		// If no next zone or function is available
		IF NextTransportData.eFunctionNumber = E_FunctionNumber.F_BEGIN_FUNCTION AND
		   Param.reNextFunctionNumber = E_FunctionNumber.F_BEGIN_FUNCTION THEN	
			// Update for this transport valid trasport parameter
			TransportParam := ZoneData.TransportControlData.TransportParam;	
		END_IF

		// If zone is occupied
		IF ZoneOccupiedSignal THEN
			// Reset clearing
			fbClearing(Run := FALSE);
			// Reset delay zone free
			fbDelayZoneFree(Run := FALSE);

			// If not status occupied
			IF NOT ZoneData.TransportControlData.Occupied THEN
				DelayDistance := TransportParam.StopDelayDistance - StoppingDistance;
				
				IF DelayDistance < 0 THEN
					DelayDistance := 0;
				END_IF
				
				// Run delay zone occupied
				fbDelayZoneOccupied(
					Run					:= TRUE,
					EncoderValueInc		:= EncoderValue,
					MaxEncoderValueInc	:= MaxEncoderValue,
					RateIncPerMM		:= 1,
					SetPoint			:= DelayDistance);

				// Set status occupied	
				IF fbDelayZoneOccupied.Q THEN
					DriveMultiTU_Run := FALSE;
					fbDelayZoneOccupied(RUN := FALSE);
					fbClearing(Run := FALSE);
					ZoneData.TransportControlData.Occupied := TRUE;
					ZoneData.TransportControlData.eTransportState := E_TransportState.MULTI_TU_OCCUPIED;
				END_IF					

			// Switch to occupied state if handover is not active
			ELSIF ZoneData.TransportControlData.eHandOverState <> E_HandOverState.ACTIVE THEN
				DriveMultiTU_Run := FALSE;
				ZoneData.TransportControlData.eTransportState := E_TransportState.MULTI_TU_OCCUPIED;
			END_IF
		
		// Zone is not occupied	
		ELSE
			// Reset delay zone occupied
			fbDelayZoneOccupied(RUN := FALSE);		

			// If status occupied
			IF ZoneData.TransportControlData.Occupied THEN
				// If handover is active
				IF ZoneData.TransportControlData.eHandOverState = E_HandOverState.ACTIVE THEN
					DelayDistance := TransportParam.ZoneEndLength - StoppingDistance;
					
					IF DelayDistance < 0 THEN
						DelayDistance := 0;
					END_IF
					
					// Run delay zone free
					fbDelayZoneFree(
						Run					:= TRUE,
						EncoderValueInc		:= EncoderValue,
						MaxEncoderValueInc	:= MaxEncoderValue,
						RateIncPerMM		:= 1,
						SetPoint			:= DelayDistance);
	
					// Restet status occupied if zone is free during handover
					IF fbDelayZoneFree.Q THEN
						fbDelayZoneFree(Run := FALSE);
						ZoneData.TransportControlData.Occupied := FALSE;
					END_IF
				ELSE
					// Switch to occupied state if handover is not active
					DriveMultiTU_Run := FALSE;
					fbDelayZoneFree(Run := FALSE);
					ZoneData.TransportControlData.eTransportState := E_TransportState.MULTI_TU_OCCUPIED;
				END_IF
	
			// Status is not occupied
			ELSE
				// Reset clearing if takeover is active
				IF ZoneData.TransportControlData.eTakeOverState = E_TakeOverState.ACTIVE THEN
					fbClearing(Run := FALSE);	
				ELSE
					// Run clearing
					fbClearing(
						Run					:= TRUE,
						EncoderValueInc		:= EncoderValue,
						MaxEncoderValueInc	:= MaxEncoderValue,
						RateIncPerMM		:= 1,
						SetPoint			:= Param.rSettings.ClearingDistance);
	
					// Switch to state free if zone is clear
					IF fbClearing.Q THEN
						DriveMultiTU_Run := FALSE;
						fbClearing(Run := FALSE);
						ZoneData.TransportControlData.NumberOfPresentTUs := 0;
						ZoneData.TransportControlData.eTransportState := E_TransportState.FREE;
					END_IF
				END_IF
			END_IF
		END_IF

(*************************************************************************
  Multi TU Occupied
*************************************************************************)
	E_TransportState.MULTI_TU_OCCUPIED:		
		// Request next zone for handover
		M_RequestNext();

		// If next zone is available
		IF NextTransportData.eFunctionNumber <> E_FunctionNumber.F_BEGIN_FUNCTION THEN
			// If handover is active
			IF ZoneData.TransportControlData.eHandOverState = E_HandOverState.ACTIVE THEN
				ZoneData.TransportControlData.eTransportState := E_TransportState.MULTI_TU;
			END_IF
		ELSE
			// Update for this transport valid trasport parameter
			TransportParam := ZoneData.TransportControlData.TransportParam;
		END_IF

		// If the occupied state needs not to be latched
		IF NOT Param.rSettings.EnableLatchOccupiedState THEN		
			// If zone is free
			IF NOT ZoneOccupiedSignal THEN
				// Run occupied free timer
				fbZoneOccupiedFreeTimer(IN := TRUE, PT := tZoneFree);

				// Zone is free without transfer
				IF fbZoneOccupiedFreeTimer.Q THEN
					fbZoneOccupiedFreeTimer(IN := FALSE);
					ZoneData.TransportControlData.Occupied := FALSE;
					TransportTrspDataReq.DeleteNextTransportData := TRUE;
	
					// Update number of present TUs
					IF ZoneData.TransportControlData.NumberOfPresentTUs > 0 THEN
						ZoneData.TransportControlData.NumberOfPresentTUs := ZoneData.TransportControlData.NumberOfPresentTUs -1;	
					END_IF			
	
					ZoneData.TransportControlData.eTransportState := E_TransportState.MULTI_TU;
				END_IF	
			ELSE
				// Reset occupied free timer
				fbZoneOccupiedFreeTimer(IN := FALSE);
			END_IF
		END_IF
				
(*************************************************************************
  Multi TU Stop
*************************************************************************)
	E_TransportState.MULTI_TU_STOP:
		// If function is started
		IF Param.rOperationState.eState = E_PositionState.STARTED THEN
			// If transport is enabled
			IF Inputs.Enable.Transport THEN		
				// If no error is active
				IF ErrorData.ErrorType <> E_ErrorType.ERROR THEN
					// If take and handover is not interrupted
					IF  ZoneData.TransportControlData.eTakeOverState <> E_TakeOverState.INTERRUPTED AND
                        ZoneData.TransportControlData.eHandOverState <> E_HandOverState.INTERRUPTED THEN
						fbZoneOccupiedFreeTimer(IN := FALSE);
						// Resume to multi TU
						ZoneData.TransportControlData.eTransportState := E_TransportState.MULTI_TU;
					END_IF
				END_IF
			END_IF
		END_IF
		
(*************************************************************************
  Simultaneous
*************************************************************************)
	E_TransportState.SIMULTANEOUS:
		// Swich to simultaneous stop if take or handover is stop or interrupted
		IF ZoneData.TransportControlData.eTakeOverState = E_TakeOverState.STOP OR 
           ZoneData.TransportControlData.eHandOverState = E_HandOverState.STOP OR
		   ZoneData.TransportControlData.eTakeOverState = E_TakeOverState.INTERRUPTED OR
		   ZoneData.TransportControlData.eHandOverState = E_HandOverState.INTERRUPTED THEN
		    DriveFeedInRun := FALSE;
			ZoneData.TransportControlData.eTransportState := E_TransportState.SIMULTANEOUS_STOP;
		END_IF	

		// If zone is physically occupied
		IF ZoneOccupiedSignal THEN
			// Reset timeout take
			fbTimeoutTake(Run := FALSE);
			// Reset delay zone free
			fbDelayZoneFree(Run := FALSE);

			// If zone is logically not occupied,
			// -> move forward until logically occupied 
			IF NOT ZoneData.TransportControlData.Occupied THEN
				// Set drive on
				DriveFeedInRun := TRUE;

				DelayDistance := TransportParam.StopDelayDistance - StoppingDistance;
				
				IF DelayDistance < 0 THEN
					DelayDistance := 0;
				END_IF
				
				// Run delay zone occupied
				fbDelayZoneOccupied(
					Run					:= TRUE,
					EncoderValueInc		:= EncoderValue,
					MaxEncoderValueInc	:= MaxEncoderValue,
					RateIncPerMM		:= 1,
					SetPoint			:= DelayDistance);

				// Set status occupied	
				IF fbDelayZoneOccupied.Q THEN
					fbDelayZoneOccupied(RUN := FALSE);
					fbClearing(Run := FALSE);
					ZoneData.TransportControlData.Occupied := TRUE;
				END_IF					
		
			// Switch to simultaneous occupied state if handover is not active
			ELSIF ZoneData.TransportControlData.eHandOverState <> E_HandOverState.ACTIVE THEN 
				DriveFeedInRun := FALSE;
				ZoneData.TransportControlData.eTransportState := E_TransportState.SIMULTANEOUS_OCCUPIED;
			ELSE
				DriveFeedInRun := FALSE;
			END_IF			
			
		// Zone is physically not occupied	
		ELSE
			// Reset delay zone occupied
			fbDelayZoneOccupied(RUN := FALSE);		

			// If zone is logically occupied
			IF ZoneData.TransportControlData.Occupied THEN
				// If handover is active
				IF ZoneData.TransportControlData.eHandOverState = E_HandOverState.ACTIVE THEN
					DelayDistance := TransportParam.ZoneEndLength - StoppingDistance;
                    DriveFeedInRun := TRUE;
					
					IF DelayDistance < 0 THEN
						DelayDistance := 0;
					END_IF
					
					// Run delay zone free
					fbDelayZoneFree(
						Run					:= TRUE,
						EncoderValueInc		:= EncoderValue,
						MaxEncoderValueInc	:= MaxEncoderValue,
						RateIncPerMM		:= 1,
						SetPoint			:= DelayDistance);
	
					// Restet status occupied if zone is free during handover
					IF fbDelayZoneFree.Q THEN
						fbDelayZoneFree(Run := FALSE);
						ZoneData.TransportControlData.Occupied := FALSE;
					END_IF
				ELSE
					// Switch to occupied state if handover is not active
					DriveFeedInRun := FALSE;
					fbDelayZoneFree(Run := FALSE);
					ZoneData.TransportControlData.eTransportState := E_TransportState.SIMULTANEOUS_OCCUPIED;
				END_IF
	
			// Zone is logically not occupied -> (Feedin)
			// adption to BCF 1.13 where this only occure if MFC is disabled
			ELSIF(NOT Param.rSettings.EnableMFC) THEN
				// Set drive on
				DriveFeedInRun := TRUE;
				
				// Timeout take monitoring
				IF Param.rSettings.TimeoutTakeDistance <> 0 THEN
					TimeoutTakeDistance := Param.rSettings.TimeoutTakeDistance;
				ELSE
					TimeoutTakeDistance := (UINT_TO_DINT(TransportParam.ZoneLength)
											- TransportParam.ZoneEndLength
											+ TransportParam.StopDelayDistance
											+ PrevTransportParam.ZoneEndLength) * TIMEOUT_TAKE_FACTOR;
				END_IF			
				
				IF TimeoutTakeDistance < 0 THEN
					TimeoutTakeDistance := 0;
				END_IF
				
				// Run timeout take
				fbTimeoutTake(
					Run					:= TRUE,
					EncoderValueInc		:= EncoderValue,
					MaxEncoderValueInc	:= MaxEncoderValue,
					SetPoint			:= TimeoutTakeDistance);
							
				// If timeout take, clear TU-data index and end feed in
				IF fbTimeoutTake.Q THEN
					// Debug message: '11-001-0095-01-1,  TU_DataIndex of implausible simultaneously takeover deleted,  TU_DataIndex = 12345,  TuID = 112233,  AssignmentID = 12345678'
					DebugMsg := '';
					DebugMsg := CONCAT(DebugMsg, F_AddDividerToSisString(Param.rSettings.ZoneName));
					DebugMsg := CONCAT(DebugMsg, ',  TU_DataIndex of implausible simultaneously takeover deleted');
					DebugMsg := CONCAT(DebugMsg, F_CreateTU_DataString(ZoneData.TransportControlData.TU_DataIndex));
					fbDebugMsg.M_SendErrorMsg(DebugMsg);
					
					DriveFeedInRun := FALSE;
					fbTimeoutTake(Run := FALSE);
					fbDelayZoneOccupied(Run := FALSE);
					M_DeleteTU_DataIndex(mSendTUR := TRUE);
					TransportTrspDataReq.DeleteNextTransportData := TRUE;
					ZoneData.TransportControlData.NumberOfPresentTUs := 0;	
	
					// If free run is enable
					IF Param.rSettings.EnableFreeRun THEN
						DriveFreeRun := TRUE;
						ZoneData.TransportControlData.eTransportState := E_TransportState.FREE_RUN;
					ELSE
						ZoneData.TransportControlData.eTransportState := E_TransportState.FREE;	
					END_IF
				END_IF
			END_IF
		END_IF
		
(*************************************************************************
  Simultaneous Occupied
*************************************************************************)
	E_TransportState.SIMULTANEOUS_OCCUPIED:		
		// If simultaneous transport is disable, switch to basic transport
		IF NOT Param.rSettings.EnableSimultaneousTransport AND
			NOT ZoneData.AddOn.Orders.EnableSimultaneousTransport THEN
			ZoneData.TransportControlData.eTransportState := E_TransportState.OCCUPIED;
		END_IF
			
		// Request prev zone for takeover
		M_RequestPrev();

		// Request next zone for handover
		M_RequestNext();

		// If next zone is available
		IF NextTransportData.eFunctionNumber <> E_FunctionNumber.F_BEGIN_FUNCTION THEN
			// If handover is active
			IF ZoneData.TransportControlData.eHandOverState = E_HandOverState.ACTIVE THEN
				ZoneData.TransportControlData.eTransportState := E_TransportState.SIMULTANEOUS;
			// Otherwise if only handover is enabled do a single handover
			ELSIF NOT Inputs.Enable.TakeOver AND Inputs.Enable.HandOver THEN
				ZoneData.TransportControlData.eTransportState := E_TransportState.HANDOVER;
			END_IF
		ELSE
			// Update for this transport valid trasport parameter
			TransportParam := ZoneData.TransportControlData.TransportParam;

			// If only handover is enabled do a single handover
			IF NOT Inputs.Enable.TakeOver AND Inputs.Enable.HandOver THEN
				ZoneData.TransportControlData.eTransportState := E_TransportState.OCCUPIED;
			END_IF
		END_IF

		// If the occupied state needs not to be latched
		IF NOT Param.rSettings.EnableLatchOccupiedState THEN	
			// If zone is free
			IF NOT ZoneOccupiedSignal THEN
				// Run occupied free timer
				fbZoneOccupiedFreeTimer(IN := TRUE, PT := tZoneFree);

				// Zone is free without transfer
				IF fbZoneOccupiedFreeTimer.Q THEN
					fbZoneOccupiedFreeTimer(IN := FALSE);
	
					// If transport is without MFC
					IF NOT Param.rSettings.EnableMFC THEN
						// Delete TU-data if it is configured
						IF Param.rSettings.DeleteTU_DataZoneFree THEN
							// debug message: '11-001-0095-01-1,  TU_DataIndex of transferless freed zone deleted,  TU_DataIndex = 5,  TuID = 000012345,  AssignmentID = 999999999'
							DebugMsg := '';
							DebugMsg := CONCAT(DebugMsg, F_AddDividerToSisString(Param.rSettings.ZoneName));
							DebugMsg := CONCAT(DebugMsg, ',  TU_DataIndex of transferless freed zone deleted');
							DebugMsg := CONCAT(DebugMsg, F_CreateTU_DataString(TU_DataIndex:= ZoneData.TransportControlData.TU_DataIndex));
							fbDebugMsg.M_SendErrorMsg(DebugMsg);
							F_DeleteTU_Data(
								TU_DataIndex 	:= ZoneData.TransportControlData.TU_DataIndex,
								NoTTC 			:= FALSE);
						END_IF
		
						M_DeleteTU_DataIndex(mSendTUR := NOT Param.rSettings.DeleteTU_DataZoneFree);
						ZoneData.TransportControlData.Occupied := FALSE;
						TransportTrspDataReq.DeleteNextTransportData := TRUE;
						ZoneData.TransportControlData.NumberOfPresentTUs := 0;				
					    DriveClearingRun:= TRUE;
						ZoneData.TransportControlData.eTransportState := E_TransportState.CLEARING;
	
					// Transport with MFC
					ELSE
						// If a TU data index is present
						IF ZoneData.TransportControlData.TU_DataIndex <> 0 THEN
							// Set error
							F_SetError(	
								ErrorType	:= E_ErrorType.ERROR,
								ErrorParam	:= '',
								ErrorMsg	:= E_ErrorConv.TU_DATA_SET_OCCUPIED_ZONE_FREE,
								ErrorData	:= ErrorData);
						ELSE
							ZoneData.TransportControlData.Occupied := FALSE;
							fbZoneOccupiedFreeTimer(IN := FALSE);
							TransportTrspDataReq.DeleteNextTransportData := TRUE;
							ZoneData.TransportControlData.NumberOfPresentTUs := 0;
	
							// If free run is enable
							IF Param.rSettings.EnableFreeRun THEN
								DriveFreeRun := TRUE;
								ZoneData.TransportControlData.eTransportState := E_TransportState.FREE_RUN;
							ELSE
								ZoneData.TransportControlData.eTransportState := E_TransportState.FREE;	
							END_IF
						END_IF
					END_IF
				END_IF
			ELSE
				// Reset occupied free timer
				fbZoneOccupiedFreeTimer(IN := FALSE);
		
				// If add TU data is configured and no TU data index is existing
				IF Param.rSettings.AddTU_Data AND ZoneData.TransportControlData.TU_DataIndex = 0 AND
					NOT Param.rSettings.EnableMultipleTU_Transition THEN
					// Insert TU-data
					ZoneData.TransportControlData.TU_DataIndex := F_InsertTU_Data(
																		eFunctionNumber := Param.reFunctionNumber,
																		ZoneNumber 		:= Param.ZoneNumber);
					// Updata data present status
					ZoneData.TransportControlData.DataPresent := ZoneData.TransportControlData.TU_DataIndex <> 0;								
					// If insert TU data is failed
					IF ZoneData.TransportControlData.TU_DataIndex = 0 THEN
						// Set error
						F_SetError(	
							ErrorType	:= E_ErrorType.ERROR,
							ErrorParam	:= '',
							ErrorMsg	:= E_ErrorConv.NO_FREE_TU_DATA_SET,
							ErrorData	:= ErrorData);
					END_IF
				END_IF
		
				// If material flow control is enabled
				IF Param.rSettings.EnableMFC THEN
					// If no TU data index is present
					IF ZoneData.TransportControlData.TU_DataIndex = 0 THEN
						// If the index is not moved to the next zone
						IF NextTransportData.rTransportControlData.eTakeOverState <> E_TakeOverState.ACTIVE THEN	
							// Set error
							F_SetError(	
								ErrorType	:= E_ErrorType.ERROR,
								ErrorParam	:= '',
								ErrorMsg	:= E_ErrorConv.TU_DATA_SET_EMPTY_ZONE_OCCUPIED,
								ErrorData	:= ErrorData);
						END_IF
					END_IF
				END_IF
			END_IF
		END_IF

(*************************************************************************
  Simultaneous Stop
*************************************************************************)
	E_TransportState.SIMULTANEOUS_STOP:		
		// Request prev zone for takeover
		M_RequestPrev();

  		// Request next zone for handover
		M_RequestNext();

		// If next zone is available
		IF NextTransportData.eFunctionNumber <> E_FunctionNumber.F_BEGIN_FUNCTION THEN
			// If function is started
			IF Param.rOperationState.eState = E_PositionState.STARTED THEN
				// If transport is enabled
				IF Inputs.Enable.Transport THEN		
					// If no error is active
					IF ErrorData.ErrorType <> E_ErrorType.ERROR THEN
						// If handover is active
						IF	ZoneData.TransportControlData.eHandOverState = E_HandOverState.ACTIVE  THEN	
							// If prev function is ready to handover 	
							IF PrevTransportData.rTransportControlData.eHandOverState = E_HandOverState.READY  THEN
								// Resume to simultaneous transport, otherwise do handover
								ZoneData.TransportControlData.eTransportState := E_TransportState.SIMULTANEOUS;
							ELSE
								ZoneData.TransportControlData.eTransportState := E_TransportState.HANDOVER;
							END_IF
						END_IF
					END_IF
				END_IF
			END_IF		
		END_IF
			
(*************************************************************************
  State Error
*************************************************************************)
ELSE
	// Set error
	F_SetError(	
		ErrorType	:= E_ErrorType.ERROR,
		ErrorParam	:= INT_TO_STRING(ZoneData.TransportControlData.eTransportState),
		ErrorMsg	:= E_ErrorConv.SOFTWARE_ERROR,
		ErrorData	:= ErrorData);	
END_CASE
END_ACTION

METHOD PROTECTED M_DeleteTU_DataIndex : BOOL
(**************************************************************************************
 * 	Application		:	BoxControl Framework
 *	Revision		:	$Revision: 475083 $
 *	Revision date	:	$Date: 2021-04-10 12:07:10 +0200 (lör, 10 apr 2021) $
 *	Last changed by	:	$Author: d7mangc $
 *	URL				:	$URL: http://almscdc.swisslog.com/repo/SWPD/Development/BoxControlFramework/20_Release/tags/R1.12.0/01_Software/BCF/BCF/JumpStart/20_Product/10_BCF/11_Conv/12_E_Functions/10_Helper/FB_TransportControl.TcPOU $
 *
 *	Purpose			:	Deletes TU-DataIndex and sends a TUR if requested and send mode selected in the settings allows sending in that case.
 *
 * ------------------------------------------------------------------------------------
 *	Copyright Swisslog [IP AG], Switzerland. All rights reserved.
 * 
 * ------------------------------------------------------------------------------------
 *	
 * 	Revision History: 
 *
 * 	VERSION			DATE			INITIALS			DESCRIPTION
 *	0.1				01.01.2001		swl					Example
 *
 **************************************************************************************)
VAR_INPUT
	mSendTUR			: BOOL; // Request to send TUR, depends on the setting eTUR_SendAllowedMode if it will be sent
END_VAR
VAR
	mIdx				: INT; //loop variable
	mDestinationList	: ARRAY [1..Conveyor.NUMBER_OF_DESTINATIONS] OF STRING(Conveyor.POSITION_STRINGLENGTH); //If TUR is to be sent, temp store for destinations for the message building
	mSendTUR_Allowed	: BOOL; //Result of checking if the sendmode allows sending of the TUR in this particular call
	mTU_DataIndex		: DINT; //local copy of the dataindex location of the TU data to be sent
END_VAR
{warning disable C0371}
IF __ISVALIDREF(ZoneData) THEN
	// If a TU-data index is existing 
	mTU_DataIndex := ZoneData.TransportControlData.TU_DataIndex;
	
	IF mTU_DataIndex <> 0 THEN
		// When TUR should be sent
		IF mSendTUR THEN
			//If the TUR was requested to be sent, first check if it should be sent according to the config of the Zone
			CASE  Param.rSettings.eTUR_SendMode OF
			E_TUR_SendModes.ALWAYS:
				mSendTUR_Allowed := TRUE;

			E_TUR_SendModes.DISABLED:
				mSendTUR_Allowed := FALSE;

			E_TUR_SendModes.DISABLE_ON_UNKNOWN_ASSIGNMENT: 
				mSendTUR_Allowed := TU_DataTable[mTU_DataIndex].AssignmentID <> Conveyor.ASSIGNMENT_ID_UNKNOWN;

			E_TUR_SendModes.DISABLE_ON_UNKNOWN_TU:
				mSendTUR_Allowed := TU_DataTable[mTU_DataIndex].TU_ID.ASCII <> Conveyor.TU_ID_UNKNOWN;

			E_TUR_SendModes.DISABLE_ON_UNKNOWN_TU_ASSIGNMENT:
				mSendTUR_Allowed := 	TU_DataTable[mTU_DataIndex].TU_ID.ASCII <> Conveyor.TU_ID_UNKNOWN
									AND TU_DataTable[mTU_DataIndex].AssignmentID <> Conveyor.ASSIGNMENT_ID_UNKNOWN;
			ELSE
				mSendTUR_Allowed := TRUE;
			END_CASE
	 		
			IF mSendTUR_Allowed THEN
				
				// Get all destinations
				FOR mIdx := 1 TO Conveyor.NUMBER_OF_DESTINATIONS DO
					IF TU_DataTable[mTU_DataIndex].Destination[mIdx].eFunctionNumber <> E_FunctionNumber.F_BEGIN_FUNCTION THEN
						mDestinationList[mIdx] := F_ReduceToAlphaNumeric(TU_DataTable[mTU_DataIndex].Destination[mIdx].PositionName);
					ELSE
						EXIT;
					END_IF
				END_FOR
				
				// Send TUR
				F_ITC_SendTUR(
					eChannelSrc				:= E_MFCS_Channel.AM,
					LastPositionName		:= F_ReduceToAlphaNumeric(FunctionRegistry[Param.reFunctionNumber].Zone[Param.ZoneNumber].ZoneName),
					TU_DataIndex			:= ZoneData.TransportControlData.TU_DataIndex,
					TU_ID					:= TU_DataTable[mTU_DataIndex].TU_ID.ASCII,
					TU_Type					:= TU_DataTable[mTU_DataIndex].DataSet.TU_Type,
					AssignmentID			:= TU_DataTable[mTU_DataIndex].AssignmentID,
					Length					:= TU_DataTable[mTU_DataIndex].DataSet.Dimension.Length,
					Width					:= TU_DataTable[mTU_DataIndex].DataSet.Dimension.Width,
					Height					:= TU_DataTable[mTU_DataIndex].DataSet.Dimension.Height,
					Weight					:= TU_DataTable[mTU_DataIndex].DataSet.Dimension.Weight,
					Orientation				:= TU_DataTable[mTU_DataIndex].DataSet.Orientation,
					TU_Parameter			:= TU_DataTable[mTU_DataIndex].DataSet.TU_Parameter,
					IO_Data					:= TU_DataTable[mTU_DataIndex].DataSet.IO_Data,
					LowerLimit				:= TU_DataTable[mTU_DataIndex].DataSet.LowerLimit,
					UpperLimit				:= TU_DataTable[mTU_DataIndex].DataSet.UpperLimit,
					Sequence				:= TU_DataTable[mTU_DataIndex].DataSet.Sequence,
					SubSequence				:= TU_DataTable[mTU_DataIndex].DataSet.SubSequence,
					SequenceSize			:= TU_DataTable[mTU_DataIndex].DataSet.SequenceSize,
					GroupID					:= TU_DataTable[mTU_DataIndex].DataSet.GroupID,
					GroupSize				:= TU_DataTable[mTU_DataIndex].DataSet.GroupSize,
					DestinationSlot         := TU_DataTable[mTU_DataIndex].DataSet.DestinationSlot,
					eReturnCode				:= E_ErrorConv.DESTINATION_NOT_REACHABLE,
					NumberOfDestinations	:= TU_DataTable[mTU_DataIndex].DataSet.NumberOfDest,
					Destination				:= mDestinationList);
			END_IF
		END_IF
		
		// Update last TU data index			
		IF ZoneData.TransportControlData.TU_DataIndex <> 0 THEN
			ZoneData.TransportControlData.LastTU_DataIndex := ZoneData.TransportControlData.TU_DataIndex;
		END_IF
		
		// Update states
		ZoneData.TransportControlData.TU_DataIndex := 0;
		ZoneData.TransportControlData.DataPresent := FALSE;
		M_DeleteTU_DataIndex := TRUE;
	END_IF
ELSE
	M_DeleteTU_DataIndex := FALSE;
END_IF
{warning restore C0371}
END_METHOD

// Moves the TU data index from previous to own zone
METHOD PROTECTED M_MoveTUdata
(**************************************************************************************
 * 	Application		:	BoxControl Framework
 *	Revision		:	$Revision: 475083 $
 *	Revision date	:	$Date: 2021-04-10 12:07:10 +0200 (lör, 10 apr 2021) $
 *	Last changed by	:	$Author: d7mangc $
 *	URL				:	$URL: http://almscdc.swisslog.com/repo/SWPD/Development/BoxControlFramework/20_Release/tags/R1.12.0/01_Software/BCF/BCF/JumpStart/20_Product/10_BCF/11_Conv/12_E_Functions/10_Helper/FB_TransportControl.TcPOU $
 *
 *	Purpose			:	Moves the TU data index from previous to own zone.
 *
 * ------------------------------------------------------------------------------------
 *	Copyright Swisslog [IP AG], Switzerland. All rights reserved.
 * 
 * ------------------------------------------------------------------------------------
 *	
 * 	Revision History: 
 *
 * 	VERSION			DATE			INITIALS			DESCRIPTION
 *	0.1				29.09.2020		swl					Example
 *
 **************************************************************************************)
VAR
  mTU_DataIndex          : DINT;
  mCurrentFunctionNumber : E_FunctionNumber;
  mCurrentZoneNumber     : INT;
END_VAR
{warning disable C0371}
// If multiple TU transition is aktive
IF Param.rSettings.EnableMultipleTU_Transition THEN
	// Move TU data index from previous to own zone
  	Transition_TU_DataIndex := F_MoveTU_DataIndex(
									eFunctionNumber := PrevTransportData.eFunctionNumber,
                                    mZoneNumber     := PrevTransportData.ZoneNumber);

	// Update number of present TUs
	ZoneData.TransportControlData.NumberOfPresentTUs := ZoneData.TransportControlData.NumberOfPresentTUs + 1;

// Else if own TU data index is free
ELSIF ZoneData.TransportControlData.TU_DataIndex = 0 THEN
	// Move TU data index from previous to own zone
	mTU_DataIndex := F_MoveTU_DataIndex(
							eFunctionNumber := PrevTransportData.eFunctionNumber,
							mZoneNumber     := PrevTransportData.ZoneNumber);

	// Update zone data
	ZoneData.TransportControlData.TU_DataIndex := mTU_DataIndex;
	ZoneData.TransportControlData.DataPresent := mTU_DataIndex <> 0;
	ZoneData.TransportControlData.NumberOfPresentTUs := 1;

	// Check if the TU data index is valid - if not, create a debug message
	IF mTU_DataIndex < 0 OR mTU_DataIndex > Conveyor.NUMBER_OF_TU_DATA THEN
		// debug message: '11-001-0095-01-1,  TU_DataIndex is out of range,  TU_DataIndex = 5000,  range = 0..1979'
		DebugMsg:= '';
		DebugMsg:= CONCAT(DebugMsg, Param.rSettings.ZoneName);
		DebugMsg:= CONCAT(DebugMsg, ',  TU_DataIndex is out of range');
		DebugMsg:= CONCAT(DebugMsg, DebugTextBlocks.TU_DATA_INDEX);
		DebugMsg:= CONCAT(DebugMsg, DINT_TO_STRING(mTU_DataIndex));
		DebugMsg:= CONCAT(DebugMsg, DebugTextBlocks.RANGE);
		DebugMsg:= CONCAT(DebugMsg, DINT_TO_STRING(Conveyor.NUMBER_OF_TU_DATA));
		fbDebugMsg.M_SendErrorMsg(DebugMsg);				  
		
	// Else if a valid TU data index is available check whether the index matches the expected position.
	// If not the TU index is incorrectly linked to multiple positions at the same time.
	ELSIF mTU_DataIndex <> 0 THEN
		mCurrentFunctionNumber := TU_Table.TU_DataTable[mTU_DataIndex].CurrentFunctionNumber;
		mCurrentZoneNumber := TU_Table.TU_DataTable[mTU_DataIndex].CurrentZoneNumber;
		
		// If function and zone number is valid
		IF mCurrentFunctionNumber <> 0 AND mCurrentZoneNumber <> 0 THEN
			// If current TU position is not previous zone
			IF mCurrentFunctionNumber <> PrevTransportData.eFunctionNumber OR mCurrentZoneNumber <> PrevTransportData.ZoneNumber THEN
				// debug message: '11-001-0095-01-1,  incorrectly linked TU_DataIndex to current TU position,  expected = 11-222-3333-44-5,  current = 99-9999-1979-01-9'
				DebugMsg:= '';
				DebugMsg:= CONCAT(DebugMsg, Param.rSettings.ZoneName);
				DebugMsg:= CONCAT(DebugMsg, ',  incorrectly linked TU_DataIndex to current TU position');
				DebugMsg:= CONCAT(DebugMsg, DebugTextBlocks.EXPECTED);
				DebugMsg:= CONCAT(DebugMsg, F_GetFunctionName(
												eFunctionNumber := PrevTransportData.eFunctionNumber,
												ZoneNumber := PrevTransportData.ZoneNumber));
				DebugMsg:= CONCAT(DebugMsg, DebugTextBlocks.CURRENT);
				DebugMsg:= CONCAT(DebugMsg, F_GetFunctionName(
												eFunctionNumber := mCurrentFunctionNumber,
												ZoneNumber := mCurrentZoneNumber));
				DebugMsg:= CONCAT(DebugMsg, F_CreateTU_DataString(mTU_DataIndex));
				fbDebugMsg.M_SendErrorMsg(DebugMsg);				  
			END_IF
		END_IF

		// Update currrent TU position
		TU_Table.TU_DataTable[mTU_DataIndex].CurrentFunctionNumber := Param.reFunctionNumber;
		TU_Table.TU_DataTable[mTU_DataIndex].CurrentZoneNumber := Param.ZoneNumber;
	END_IF

ELSE
	// Own TU data index is already used
	mTU_DataIndex := ZoneData.TransportControlData.TU_DataIndex;

	// Set error TU data index is not free
	F_SetError(
		ErrorType := E_ErrorType.ERROR,
		ErrorParam:= CONCAT('TU-DataIndex = ', DINT_TO_STRING(mTU_DataIndex)),
		ErrorMsg  := E_ErrorConv.TU_DATA_INDEX_NOT_FREE,
		ErrorData := ErrorData);
	
	// debug message: '11-001-0095-01-1,  own TU data index not free,  TU_DataIndex = 12345,  TuID = 112233,  AssignmentID = 12345678'
	DebugMsg:= '';
	DebugMsg:= CONCAT(DebugMsg, Param.rSettings.ZoneName);
	DebugMsg:= CONCAT(DebugMsg, ',  own TU data index not free');
	DebugMsg:= CONCAT(DebugMsg, F_CreateTU_DataString(mTU_DataIndex));
	fbDebugMsg.M_SendErrorMsg(DebugMsg);				  
	
	// Update number of present TUs
	ZoneData.TransportControlData.NumberOfPresentTUs := 1;
END_IF
{warning restore C0371}
END_METHOD

// Requests the routing service to retrieve next partner
METHOD PROTECTED M_RequestNext
(**************************************************************************************
 *  Application     :   BoxControl Framework
 *  Revision date   :   $Date: 2021-04-10 12:07:10 +0200 (lör, 10 apr 2021) $
 *  Author          :   CDC
 * ------------------------------------------------------------------------------------
 *  © Swisslog AG
 *  Swisslog is not liable for any usage of this source code that is not agreed 
 *  on between Swisslog and the other party. The mandatory legal liability remains 
 *  unaffected.
 * ------------------------------------------------------------------------------------
 *  Revision History: 
 *
 *  VERSION DATE         INITIALS     DESCRIPTION
 *  0.0     DD.MM.YYYY   (name)       (explain customized modifications)
 *
 **************************************************************************************)
VAR_INPUT
END_VAR
{warning disable C0371}
// If no next zone or function is available
IF NextTransportData.eFunctionNumber = E_FunctionNumber.F_BEGIN_FUNCTION AND
   Param.reNextFunctionNumber = E_FunctionNumber.F_BEGIN_FUNCTION THEN	
	fbRoutingServiceRetry(IN := FALSE);
	TransportTrspDataReq.RequestNextTransportData := TRUE;

// If the routing update is enable	
ELSIF Param.rSettings.EnableRoutingUpdate THEN
	// If the next function ist not fix
	IF Param.reSetFuncNextFuncNumber = E_FunctionNumber.F_BEGIN_FUNCTION
	   AND NOT NextTransportData.rTransportControlData.TransportActive THEN
		// If the transport does not start in a reasonable time, initiate routing update
		IF ZoneData.TransportControlData.eHandOverState = E_HandOverState.IDLE OR
		   ZoneData.TransportControlData.eHandOverState = E_HandOverState.READY THEN
			fbRoutingServiceRetry(IN := TRUE, PT := RECALL_SERVICE_TIMEOUT);
			IF fbRoutingServiceRetry.Q THEN
				fbRoutingServiceRetry(IN := FALSE);
				TransportTrspDataReq.DeleteNextTransportData := TRUE;
				TransportTrspDataReq.RequestNextTransportData := TRUE;
			END_IF
		ELSE
			fbRoutingServiceRetry(IN := FALSE);
		END_IF
	ELSE
		fbRoutingServiceRetry(IN := FALSE);
	END_IF
END_IF
{warning restore C0371}
END_METHOD

// Requests the merging service to retrieve prev partner
METHOD PROTECTED M_RequestPrev
(**************************************************************************************
 *  Application     :   BoxControl Framework
 *  Revision date   :   $Date: 2021-04-10 12:07:10 +0200 (lör, 10 apr 2021) $
 *  Author          :   CDC
 * ------------------------------------------------------------------------------------
 *  © Swisslog AG
 *  Swisslog is not liable for any usage of this source code that is not agreed 
 *  on between Swisslog and the other party. The mandatory legal liability remains 
 *  unaffected.
 * ------------------------------------------------------------------------------------
 *  Revision History: 
 *
 *  VERSION DATE         INITIALS     DESCRIPTION
 *  0.0     DD.MM.YYYY   (name)       (explain customized modifications)
 *
 **************************************************************************************)
VAR_INPUT
END_VAR
{warning disable C0371}
// If no previous zone or function is available
IF PrevTransportData.eFunctionNumber = E_FunctionNumber.F_BEGIN_FUNCTION AND
   Param.rePrevFunctionNumber = E_FunctionNumber.F_BEGIN_FUNCTION THEN	
	fbMergingServiceRetry(IN := FALSE);
	TransportTrspDataReq.RequestPrevTransportData := TRUE;


// If the previous function ist not fix
ELSIF Param.reSetFuncPrevFuncNumber = E_FunctionNumber.F_BEGIN_FUNCTION
   AND NOT PrevTransportData.rTransportControlData.TransportActive THEN
	// If the transport does not start in a reasonable time, initiate merging update
	IF ZoneData.TransportControlData.eTakeOverState = E_TakeOverState.IDLE OR
	   ZoneData.TransportControlData.eTakeOverState = E_TakeOverState.READY THEN
		fbMergingServiceRetry(IN := TRUE, PT := RECALL_SERVICE_TIMEOUT);
		IF fbMergingServiceRetry.Q THEN
			fbMergingServiceRetry(IN := FALSE);
			TransportTrspDataReq.DeletePrevTransportData := TRUE;
			TransportTrspDataReq.RequestPrevTransportData := TRUE;
		END_IF
	END_IF
END_IF
{warning restore C0371}
END_METHOD

METHOD M_SelectSensor : BOOL
(**************************************************************************************
 *  Application     :   BoxControl Framework
 *  Revision date   :   $Date: 2021-04-10 12:07:10 +0200 (lör, 10 apr 2021) $
 *  Author          :   CDC
 * ------------------------------------------------------------------------------------
 *  © Swisslog AG
 *  Swisslog is not liable for any usage of this source code that is not agreed 
 *  on between Swisslog and the other party. The mandatory legal liability remains 
 *  unaffected.
 * ------------------------------------------------------------------------------------
 *  Revision History: 
 *
 *  VERSION DATE         INITIALS     DESCRIPTION
 *  0.0     DD.MM.YYYY   (name)       (explain customized modifications)
 *
 **************************************************************************************)
VAR_INPUT
END_VAR
{warning disable C0371}
IF ZoneData.AddOn.Orders.UseOwnSensor OR NOT Param.rSettings.EnableAddOnSensor THEN
    ZoneOccupiedSignal := ZoneOccupied;
ELSE
    ZoneOccupiedSignal := ZoneData.AddOn.Orders.AddOnSensor;
END_IF
{warning restore C0371}
END_METHOD

// Starts the tracking of the leading edge arriving from prev zone
METHOD PROTECTED M_StartPositionTracking
(**************************************************************************************
 *  Application     :   BoxControl Framework
 *  Revision date   :   $Date: 2021-04-10 12:07:10 +0200 (lör, 10 apr 2021) $
 *  Author          :   CDC
 * ------------------------------------------------------------------------------------
 *  © Swisslog AG
 *  Swisslog is not liable for any usage of this source code that is not agreed 
 *  on between Swisslog and the other party. The mandatory legal liability remains 
 *  unaffected.
 * ------------------------------------------------------------------------------------
 *  Revision History: 
 *
 *  VERSION DATE         INITIALS     DESCRIPTION
 *  0.0     DD.MM.YYYY   (name)       (explain customized modifications)
 *
 **************************************************************************************)
VAR
	PresetDistance     			: DINT; // Present distance for tracking leading edge
END_VAR

// Set preset distance based on available previous position data	
IF PrevTransportData.rTransportControlData.TU_LeadingEdgePos <> 0 THEN
	PresetDistance := -(UINT_TO_DINT(PrevTransportParam.ZoneLength) - PrevTransportData.rTransportControlData.TU_LeadingEdgePos);
ELSE
	PresetDistance := -(UINT_TO_DINT(PrevTransportParam.ZoneEndLength) - PrevTransportParam.StopDelayDistance);
END_IF

// Start tracking 
fbTrackingLeadingEdge(Run := FALSE);

fbTrackingLeadingEdge(Run	:= TRUE,
		EncoderValueInc 	:= EncoderValue,
		MaxEncoderValueInc	:= MaxEncoderValue,
		RateIncPerMM		:= 1,
		SetPoint			:= UINT_TO_DINT(16#FFFF),
		StartPoint			:= PresetDistance);
END_METHOD

// Calculates the distance, the TU must at least travel to be considered plausible
METHOD PROTECTED M_TakeoverPlausibleDistance : DINT
(**************************************************************************************
 *  Application     :   BoxControl Framework
 *  Revision date   :   $Date: 2021-04-10 12:07:10 +0200 (lör, 10 apr 2021) $
 *  Author          :   CDC
 * ------------------------------------------------------------------------------------
 *  © Swisslog AG
 *  Swisslog is not liable for any usage of this source code that is not agreed 
 *  on between Swisslog and the other party. The mandatory legal liability remains 
 *  unaffected.
 * ------------------------------------------------------------------------------------
 *  Revision History: 
 *
 *  VERSION DATE         INITIALS     DESCRIPTION
 *  0.0     DD.MM.YYYY   (name)       (explain customized modifications)
 *
 **************************************************************************************)
VAR
	Temp		: DINT		:= 0;
END_VAR

// valid value given from config -> use this
IF Param.rSettings.TakeoverPlausibilityDistance <> 0 THEN
	M_TakeoverPlausibleDistance := Param.rSettings.TakeoverPlausibilityDistance;
	RETURN;
END_IF

// no, calculate it:
// distance between TU's leading edge to the border of the prev zone 
Temp:= PrevTransportParam.ZoneEndLength - PrevTransportParam.StopDelayDistance;

// adding the distance from begin of own zone to the sensor
Temp:= Temp + UINT_TO_DINT(TransportParam.ZoneLength) - TransportParam.ZoneEndLength;

// return reduced value to give space for tolerance
M_TakeoverPlausibleDistance:= Temp - DIST_TO_OCCUPIED;
END_METHOD

END_FUNCTION_BLOCK

(* stored: Version 1.1.0.1, ProductVersion 3.1.4024.9
   POU FB_TransportControl: Id {b402116b-65a1-4b4b-bdcc-6610068ed1bb}, SpecialFunc None
   Action A_Brake: Id {8bc977f7-2385-409e-a16c-51264030fcc8}
   Action A_HandOverState: Id {17832d94-ca66-48b7-8b6e-06f5c48311dd}
   Action A_Init: Id {dd49f579-06d8-455c-8903-1535dbca12f3}
   Action A_InputMapping: Id {0f804f75-256e-44ea-a1f0-1d0c23f05634}
   Action A_JamAutoReset: Id {d301aacc-851d-4bb4-997f-0a21c9463081}
   Action A_OutputMapping: Id {be78205a-8bc0-494c-ad0d-4ea7bd67489b}
   Action A_PositionTracking: Id {2a872687-daae-4b91-b8a5-b6392160b835}
   Action A_ShortZoneRestart: Id {46fae7f7-7acc-4943-8824-2601312d8a04}
   Action A_TakeOverState: Id {3ba99b51-9909-435a-8ae7-10d081ab7270}
   Action A_TransportState: Id {d3af210a-698d-4e72-9fc7-c2ba2843e98b}
   Method M_DeleteTU_DataIndex: Id {3f8c49b0-f47c-4916-aad5-8038f95e220c}
   Method M_MoveTUdata: Id {d17bde12-6418-4bd7-b590-b75b64dfcbf8}
   Method M_RequestNext: Id {2c37c848-efb9-4442-8d76-2328c143fa92}
   Method M_RequestPrev: Id {f4486108-8078-4ff0-ae47-01e4ca68e476}
   Method M_SelectSensor: Id {6ff5eb84-281c-4ff9-8db2-a56130814bcb}
   Method M_StartPositionTracking: Id {523fa34d-d115-4843-9676-8b4ef2e97ecc}
   Method M_TakeoverPlausibleDistance: Id {e1df1950-bac4-46f8-95d5-eafbd9ea500a} *)
